{attribute 'GeneratedUsingTerminal: EK1100-0000-0018'}
{attribute addProperty BoxType "EK1100-0000-0018"}
{attribute addProperty Id "Beckhoff_ER3xxxEK1122Beckhoff_ER3xxxEK1122_FC5AAA23522"}
{attribute addProperty CRC "3189414439"}
{attribute addProperty Size "522"}
TYPE Beckhoff_ER3xxx_BE1A9A27 EXTENDS EK1100_1FC0878B :
STRUCT
	{attribute addProperty Name "Beckhoff_ER3xxxEK1122"}
	{attribute addProperty PreviousPort "Beckhoff ER3xxx : B"}
	Beckhoff_ER3xxxEK1122 : Beckhoff_ER3xxxEK1122_FC5AAA23;
END_STRUCT
END_TYPE

(* stored: Version 1.2.0.0, ProductVersion 3.1.4024.9
   DUT Beckhoff_ER3xxx_BE1A9A27: Id {3c52b1bf-35a7-44ec-a578-1682bf61520b} *)
